// TIA Portal V17 export
// export: Created 2025-03-07T09:19:16.0197324Z, ExportSetting WithDefaults, DisplayName Totally Integrated Automation Portal, DisplayVersion V17 Update 8, DisplayName TIA Portal Openness, DisplayVersion V17 Update 8, DisplayName TIA Portal Version Control Interface, DisplayVersion V17, DisplayName SINAMICS Startdrive Advanced, DisplayVersion V17 SP2, DisplayName SINAMICS Startdrive G110M, G120, G120C, G120D, G120P, G115D, DisplayVersion V17 SP2, DisplayName SINAMICS Startdrive G130, G150, S120, S150, SINAMICS MV, S210, DisplayVersion V17 SP2, DisplayName STEP 7 Professional, DisplayVersion V17 Update 8, DisplayName SINUMERIK ONE STEP 7 Toolbox, DisplayVersion V17 Update 12, DisplayName SINUMERIK 840D sl STEP 7 Toolbox, DisplayVersion V17 Update 12, DisplayName STEP 7 Safety, DisplayVersion V17 Update 6, DisplayName WinCC Advanced, DisplayVersion V17 Update 8
DATA_BLOCK "DB7214_CYCLE_TIMES"   // DB7214
{ S7_Optimized_Access := 'FALSE'; DB_Accessible_From_OPC_UA := 'FALSE' }
AUTHOR : ETXETAR
VERSION : 1.0
// stored: AutoNumber false, DBAccessibleFromOPCUA false, DBAccessibleFromWebserver true, IsOnlyStoredInLoadMemory false, IsWriteProtectedInAS false
   VAR RETAIN
      U01_PART_TO_PART_CYCLE_START : Bool := FALSE;   // UNIT 01 PART TO PART CYCLE START
      U01_PART_TO_PART_CYCLE_END : Bool := FALSE;   // UNIT 01 PART TO PART CYCLE END
      U01_STA_1_CYCLE_START : Bool := FALSE;   // UNIT 01 STATION 1 CYCLE START
      U01_STA_1_CYCLE_END : Bool := FALSE;   // UNIT 01 STATION 1 CYCLE END
      U01_STA_2_CYCLE_START : Bool := FALSE;   // UNIT 01 STATION 2 CYCLE START
      U01_STA_2_CYCLE_END : Bool := FALSE;   // UNIT 01 STATION 2 CYCLE END
      U01_STA_3_CYCLE_START : Bool := FALSE;   // UNIT 01 STATION 3 CYCLE START
      U01_STA_3_CYCLE_END : Bool := FALSE;   // UNIT 01 STATION 3 CYCLE END
      U01_STA_4_CYCLE_START : Bool := FALSE;   // UNIT 01 STATION 4 CYCLE START
      U01_STA_4_CYCLE_END : Bool := FALSE;   // UNIT 01 STATION 4 CYCLE END
      U01_LOAD_CYCLE_START : Bool := FALSE;   // UNIT 01 LOAD CYCLE START
      U01_LOAD_CYCLE_END : Bool := FALSE;   // UNIT 01 LOAD CYCLE END
      U01_UNLOAD_CYCLE_START : Bool := FALSE;   // UNIT 01 UNLOAD CYCLE START
      U01_UNLOAD_CYCLE_END : Bool := FALSE;   // UNIT 01 UNLOAD CYCLE END
      U02_PART_TO_PART_CYCLE_START : Bool := FALSE;   // UNIT 02 PART TO PART CYCLE START
      U02_PART_TO_PART_CYCLE_END : Bool := FALSE;   // UNIT 02 PART TO PART CYCLE END
      U02_STA_1_CYCLE_START : Bool := FALSE;   // UNIT 02 STATION 1 CYCLE START
      U02_STA_1_CYCLE_END : Bool := FALSE;   // UNIT 02 STATION 1 CYCLE END
      U02_STA_2_CYCLE_START : Bool := FALSE;   // UNIT 02 STATION 2 CYCLE START
      U02_STA_2_CYCLE_END : Bool := FALSE;   // UNIT 02 STATION 2 CYCLE END
      U02_STA_3_CYCLE_START : Bool := FALSE;   // UNIT 02 STATION 3 CYCLE START
      U02_STA_3_CYCLE_END : Bool := FALSE;   // UNIT 02 STATION 3 CYCLE END
      U02_STA_4_CYCLE_START : Bool := FALSE;   // UNIT 02 STATION 4 CYCLE START
      U02_STA_4_CYCLE_END : Bool := FALSE;   // UNIT 02 STATION 4 CYCLE END
      U02_LOAD_CYCLE_START : Bool := FALSE;   // UNIT 02 LOAD CYCLE START
      U02_LOAD_CYCLE_END : Bool := FALSE;   // UNIT 02 LOAD CYCLE END
      U02_UNLOAD_CYCLE_START : Bool := FALSE;   // UNIT 02 UNLOAD CYCLE START
      U02_UNLOAD_CYCLE_END : Bool := FALSE;   // UNIT 02 UNLOAD CYCLE END
      TARGET_CYCLE_TIME : Int := 1200;   // TARGET CYCLE TIME
      PULSE : Bool := FALSE;   // PULSE
      PULSE1 : Bool := FALSE;   // PULSE 1
      PULSE2 : Bool := FALSE;   // PULSE 2
      PULSE3 : Bool := FALSE;   // PULSE 3
      PULSE4 : Bool := FALSE;   // PULSE 4
      PULSE5 : Bool := FALSE;   // PULSE 5
      PULSE6 : Bool := FALSE;   // PULSE 6
      PULSE7 : Bool := FALSE;   // PULSE 7
      PULSE8 : Bool := FALSE;   // PULSE 8
      PULSE9 : Bool := FALSE;   // PULSE 9
      PULSE10 : Bool := FALSE;   // PULSE 10
      PULSE11 : Bool := FALSE;   // PULSE 11
      PULSE12 : Bool := FALSE;   // PULSE 12
      PULSE13 : Bool := FALSE;   // PULSE 13
      PULSE14 : Bool := FALSE;   // PULSE 14
      PULSE15 : Bool := FALSE;   // PULSE 15
      PULSE16 : Bool := FALSE;   // PULSE 16
      PULSE17 : Bool := FALSE;   // PULSE 17
      PULSE18 : Bool := FALSE;   // PULSE 18
      PULSE19 : Bool := FALSE;   // PULSE 19
      PULSE20 : Bool := FALSE;   // PULSE 20
      PULSE21 : Bool := FALSE;   // PULSE 21
      PULSE22 : Bool := FALSE;   // PULSE 22
      PULSE23 : Bool := FALSE;   // PULSE 23
      PULSE24 : Bool := FALSE;   // PULSE 24
      PULSE25 : Bool := FALSE;   // PULSE 25
      PULSE26 : Bool := FALSE;   // PULSE 26
      PULSE27 : Bool := FALSE;   // PULSE 27
      PULSE28 : Bool := FALSE;   // PULSE 28
      PULSE29 : Bool := FALSE;   // PULSE 29
      PULSE30 : Bool := FALSE;   // PULSE 30
   END_VAR
BEGIN
END_DATA_BLOCK
